TYPE INTERNAL _EcUnion :
UNION
	iComponent	: I_FatComponent;
	iEntity		: I_EntityNode;
END_UNION
END_TYPE

(* stored: Version 1.1.0.1
   DUT _EcUnion: Id {03758be6-2b89-43ee-b6ee-40fda7565e5b} *)
